{attribute 'GeneratedUsingTerminal: EL1502-0000-0018'}
{attribute addProperty BoxType "EL1502-0000-0018"}
{attribute addProperty Id "CNT_InputsAT %I*CNT_Inputs_B6C38E7112CNT_OutputsAT %Q*CNT_Outputs_458039AE8WcStateAT %I*WcState_9091E0EB2InfoDataAT %I*InfoData_32EB74EA10"}
{attribute addProperty CRC "369962764"}
{attribute addProperty Size "32"}
TYPE EL1502_160D2F0C :
STRUCT
	{attribute addProperty Name "CNT_Inputs"}
	CNT_Inputs : CNT_Inputs_B6C38E71;
	{attribute addProperty Name "CNT_Outputs"}
	CNT_Outputs : CNT_Outputs_458039AE;
	{attribute addProperty Name "WcState"}
	WcState : WcState_9091E0EB;
	{attribute addProperty Name "InfoData"}
	InfoData : InfoData_32EB74EA;
END_STRUCT
END_TYPE

(* stored: Version 1.2.0.0, ProductVersion 3.1.4024.9
   DUT EL1502_160D2F0C: Id {117b4877-b08e-4d38-a62e-d24c901e8e86} *)
